(* Logix 5000 project; controller ToyPlant Emulate 5570 rev 30.12; software revision 30.00 *)

TASK MainTask (continuous, watchdog 500 ms) : MainProgram

MODULES
   Local : Emulate 5570 (ICP 2, rev 30.12)
      VIRTUAL_INPUTS : vendor 1 type 0 code 15 (ICP 3, rev 1.1, Output RPI 50 ms)
END_MODULES

PROGRAM MainProgram   (* main routine MainRoutine *)
VAR
   Action_000 : SFC_ACTION := (Status := 16#0020_0000, PauseTimer := 1, Count := 1);
   Action_001 : SFC_ACTION := (Status := 16#c020_0000, A := 1, Q := 1, PauseTimer := 1, Count := 2);
   Action_002 : SFC_ACTION := (Status := 16#0020_0000, PauseTimer := 1, Count := 1);
   Action_003 : SFC_ACTION := (Status := 16#0020_0000, PauseTimer := 1, Count := 1);
   Action_004 : SFC_ACTION := (Status := 16#0020_0000, PauseTimer := 1, Count := 1);
   Action_005 : SFC_ACTION := (Status := 16#0020_0000, PauseTimer := 1, Count := 1);
   Action_006 : SFC_ACTION := (Status := 16#0020_0000, PauseTimer := 1, Count := 1);
   Action_007 : SFC_ACTION := (Status := 16#0020_0000, PauseTimer := 1, Count := 1);
   Action_008 : SFC_ACTION := (Status := 16#0020_0000, PauseTimer := 1, Count := 1);
   StartEnsamble : ALIAS FOR Local:3:I.Data[1].0;
   Step_000 : SFC_STEP := (Status := 16#a820_0201, X := 1, SA := 1, DN := 1, PauseTimer := 1, T := 31632, TMax := 31632, Count := 2);
   Step_001 : SFC_STEP := (Status := 16#0820_0001, DN := 1, PauseTimer := 1, T := 2120, TMax := 2120, Count := 1);
   Step_002 : SFC_STEP := (Status := 16#0820_0001, DN := 1, PauseTimer := 1, T := 6321, TMax := 6321, Count := 1);
   Step_003 : SFC_STEP := (Status := 16#0820_0001, DN := 1, PauseTimer := 1, T := 741, TMax := 741, Count := 1);
   Step_004 : SFC_STEP := (Status := 16#0820_0001, DN := 1, PauseTimer := 1, T := 933, TMax := 933, Count := 1);
   Step_005 : SFC_STEP := (Status := 16#0820_0001, DN := 1, PauseTimer := 1, T := 527, TMax := 527, Count := 1);
   TimerChasis : FBD_TIMER := (TimerEnable := 1, PRE := 700, ACC := 720, EN := 1, DN := 1);
   TimerPuertaAbierta : FBD_TIMER := (TimerEnable := 1, PRE := 900, ACC := 912, EN := 1, DN := 1);
   TimerPuertaCerrada : FBD_TIMER := (TimerEnable := 1, PRE := 500, ACC := 500, EN := 1, DN := 1);
   Tran_000 : BOOL;
   Tran_001 : BOOL := 1;
   Tran_002 : BOOL := 1;
   Tran_003 : BOOL := 1;
   Tran_004 : BOOL := 1;
   Tran_005 : BOOL := 1;
END_VAR
VAR_OUTPUT
   CerrarPuertaMoto : BOOL := 1; {access Read Only}
   Chasis_0 : BOOL := 1;
   Chasis_1 : BOOL := 1;
   RuedaDelantera_0 : BOOL := 1;
   RuedaDelantera_1 : BOOL := 1;
   RuedaDelantera_2 : BOOL := 1;
   RuedaTrasera_0 : BOOL := 1;
   RuedaTrasera_1 : BOOL := 1;
   RuedaTrasera_2 : BOOL := 1;
END_VAR
VAR_INPUT
   Sensor_RuedaDelantera1 : BOOL;
   Sensor_RuedaDelantera2 : BOOL;
   Sensor_RuedaTrasera1 : BOOL;
   Sensor_RuedaTrasera2 : BOOL;
   SensorChasis : BOOL;
END_VAR

ROUTINE MainRoutine   (* sequential function chart *)
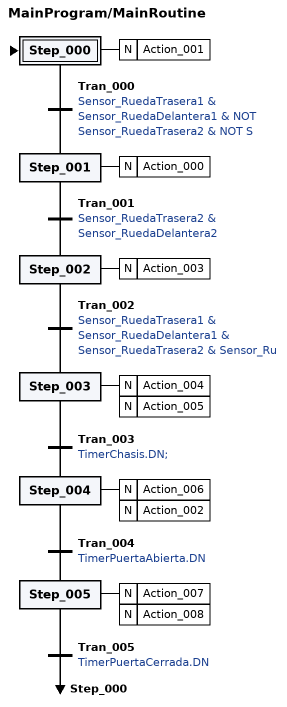
   INITIAL_STEP Step_000:
      ACTION Action_001 (N):
         CerrarPuertaMoto := 1;
      END_ACTION
   END_STEP
   TRANSITION Tran_000 FROM Step_000 TO Step_001
      := Sensor_RuedaTrasera1 & Sensor_RuedaDelantera1 & NOT Sensor_RuedaTrasera2 & NOT Sensor_RuedaDelantera2 & CerrarPuertaMoto
         
   END_TRANSITION
   STEP Step_001:
      ACTION Action_000 (N):
         RuedaDelantera_1 := 1;
         RuedaTrasera_1 := 1;
      END_ACTION
   END_STEP
   TRANSITION Tran_001 FROM Step_001 TO Step_002
      := Sensor_RuedaTrasera2 & Sensor_RuedaDelantera2
         
   END_TRANSITION
   STEP Step_002:
      ACTION Action_003 (N):
         RuedaTrasera_0 := 1;
         RuedaDelantera_0 := 1;
      END_ACTION
   END_STEP
   TRANSITION Tran_002 FROM Step_002 TO Step_003
      := Sensor_RuedaTrasera1 & Sensor_RuedaDelantera1 & Sensor_RuedaTrasera2 & Sensor_RuedaDelantera2 & SensorChasis
   END_TRANSITION
   STEP Step_003:
      ACTION Action_004 (N):
         Chasis_1 := 1;
      END_ACTION
      ACTION Action_005 (N):
         TimerChasis.TimerEnable := 1;
         TONR(TimerChasis);
         TimerChasis.PRE := 700;
         
      END_ACTION
   END_STEP
   TRANSITION Tran_003 FROM Step_003 TO Step_004
      := TimerChasis.DN;
   END_TRANSITION
   STEP Step_004:
      ACTION Action_006 (N):
         RuedaTrasera_2 := 1;
         RuedaDelantera_2 := 1;
      END_ACTION
      ACTION Action_002 (N):
         TimerPuertaAbierta.TimerEnable := 1;
         TONR(TimerPuertaAbierta);
         TimerPuertaAbierta.PRE := 900;
         
      END_ACTION
   END_STEP
   TRANSITION Tran_004 FROM Step_004 TO Step_005
      := TimerPuertaAbierta.DN
   END_TRANSITION
   STEP Step_005:
      ACTION Action_007 (N):
         CerrarPuertaMoto := 0;
         RuedaTrasera_0 := 1;
         RuedaDelantera_0 := 1;
         Chasis_0 :=1;
      END_ACTION
      ACTION Action_008 (N):
         TimerPuertaCerrada.TimerEnable := 1;
         TONR(TimerPuertaCerrada);
         TimerPuertaCerrada.PRE := 500;
         
      END_ACTION
   END_STEP
   TRANSITION Tran_005 FROM Step_005 TO Step_000
      := TimerPuertaCerrada.DN
   END_TRANSITION
END_ROUTINE
END_PROGRAM
